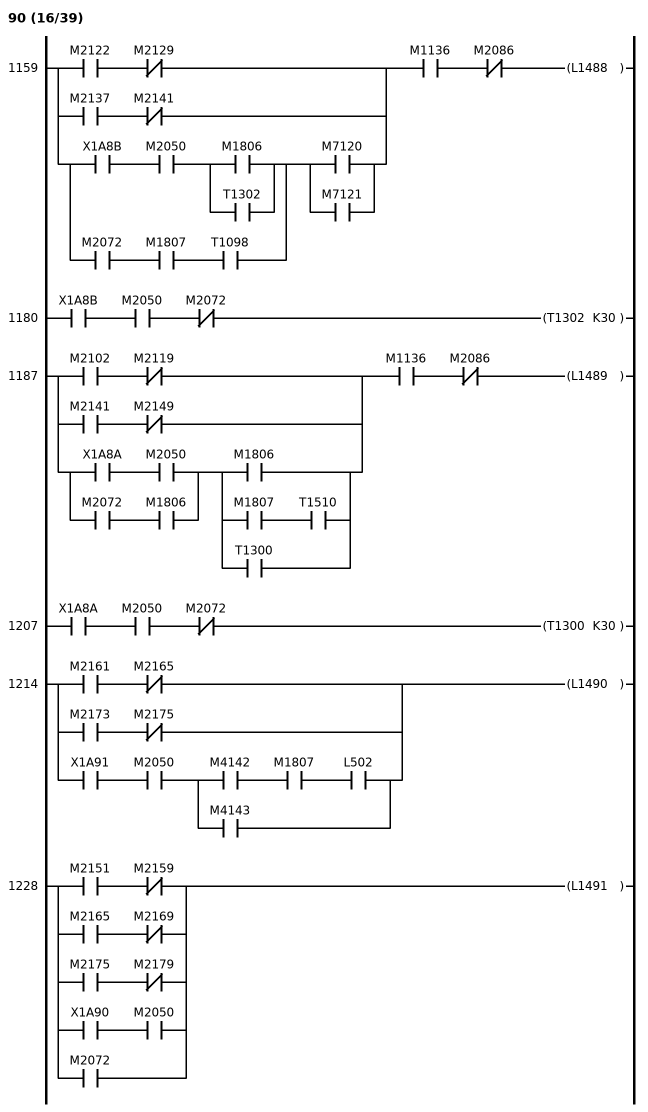
1159  LD      M2122
      ANI     M2129
      LD      M2137
      ANI     M2141
      ORB
      LD      X1A8B
      AND     M2050
      LD      M1806
      OR      T1302
      ANB
      LD      M2072
      AND     M1807
      AND     T1098
      ORB
      LD      M7120
      OR      M7121
      ANB
      ORB
      AND     M1136
      ANI     M2086
      OUT     L1488
1180  LD      X1A8B
      AND     M2050
      ANI     M2072
      OUT     T1302 K30
1187  LD      M2102
      ANI     M2119
      LD      M2141
      ANI     M2149
      ORB
      LD      X1A8A
      AND     M2050
      LD      M2072
      AND     M1806
      ORB
      LD      M1806
      LD      M1807
      AND     T1510
      ORB
      OR      T1300
      ANB
      ORB
      AND     M1136
      ANI     M2086
      OUT     L1489
1207  LD      X1A8A
      AND     M2050
      ANI     M2072
      OUT     T1300 K30
1214  LD      M2161
      ANI     M2165
      LD      M2173
      ANI     M2175
      ORB
      LD      X1A91
      AND     M2050
      LD      M4142
      AND     M1807
      AND     L502
      OR      M4143
      ANB
      ORB
      OUT     L1490
1228  LD      M2151
      ANI     M2159
      LD      M2165
      ANI     M2169
      ORB
      LD      M2175
      ANI     M2179
      ORB
      LD      X1A90
      AND     M2050
      ORB
      OR      M2072
      OUT     L1491
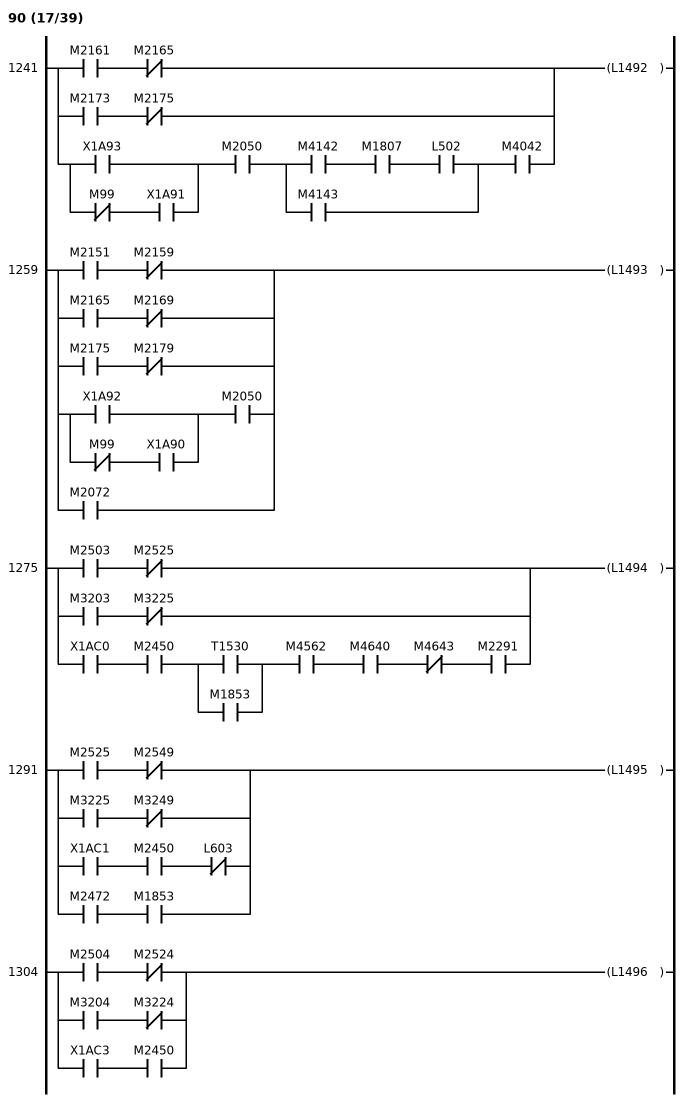
1241  LD      M2161
      ANI     M2165
      LD      M2173
      ANI     M2175
      ORB
      LD      X1A93
      LDI     M99
      AND     X1A91
      ORB
      AND     M2050
      LD      M4142
      AND     M1807
      AND     L502
      OR      M4143
      ANB
      AND     M4042
      ORB
      OUT     L1492
1259  LD      M2151
      ANI     M2159
      LD      M2165
      ANI     M2169
      ORB
      LD      M2175
      ANI     M2179
      ORB
      LD      X1A92
      LDI     M99
      AND     X1A90
      ORB
      AND     M2050
      ORB
      OR      M2072
      OUT     L1493
1275  LD      M2503
      ANI     M2525
      LD      M3203
      ANI     M3225
      ORB
      LD      X1AC0
      AND     M2450
      LD      T1530
      OR      M1853
      ANB
      AND     M4562
      AND     M4640
      ANI     M4643
      AND     M2291
      ORB
      OUT     L1494
1291  LD      M2525
      ANI     M2549
      LD      M3225
      ANI     M3249
      ORB
      LD      X1AC1
      AND     M2450
      ANI     L603
      ORB
      LD      M2472
      AND     M1853
      ORB
      OUT     L1495
1304  LD      M2504
      ANI     M2524
      LD      M3204
      ANI     M3224
      ORB
      LD      X1AC3
      AND     M2450
      ORB
      OUT     L1496
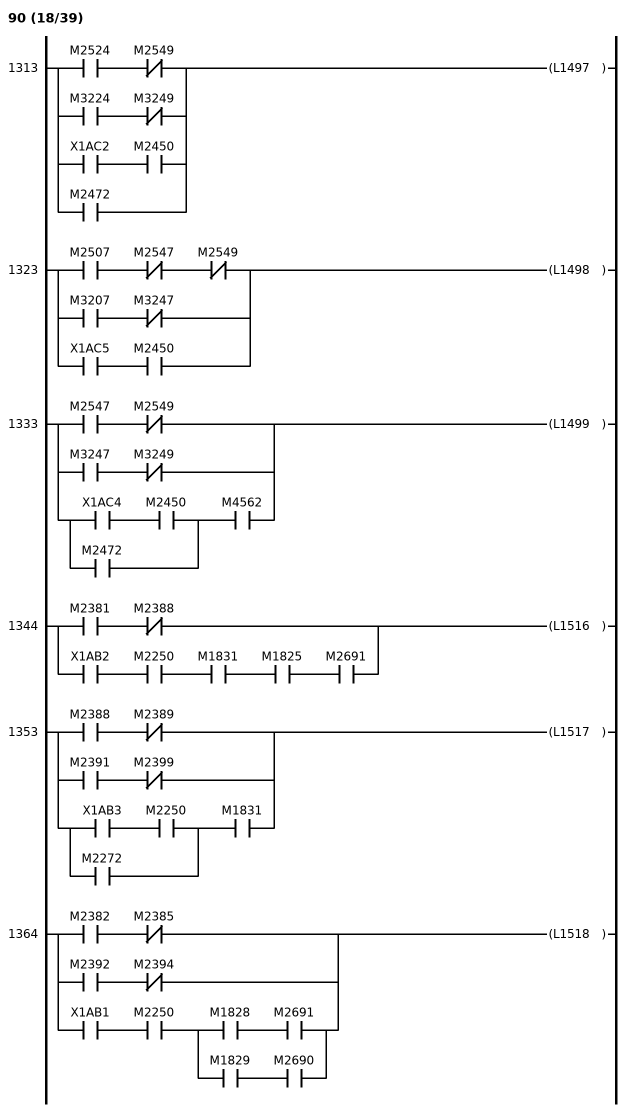
1313  LD      M2524
      ANI     M2549
      LD      M3224
      ANI     M3249
      ORB
      LD      X1AC2
      AND     M2450
      ORB
      OR      M2472
      OUT     L1497
1323  LD      M2507
      ANI     M2547
      ANI     M2549
      LD      M3207
      ANI     M3247
      ORB
      LD      X1AC5
      AND     M2450
      ORB
      OUT     L1498
1333  LD      M2547
      ANI     M2549
      LD      M3247
      ANI     M3249
      ORB
      LD      X1AC4
      AND     M2450
      OR      M2472
      AND     M4562
      ORB
      OUT     L1499
1344  LD      M2381
      ANI     M2388
      LD      X1AB2
      AND     M2250
      AND     M1831
      AND     M1825
      AND     M2691
      ORB
      OUT     L1516
1353  LD      M2388
      ANI     M2389
      LD      M2391
      ANI     M2399
      ORB
      LD      X1AB3
      AND     M2250
      OR      M2272
      AND     M1831
      ORB
      OUT     L1517
1364  LD      M2382
      ANI     M2385
      LD      M2392
      ANI     M2394
      ORB
      LD      X1AB1
      AND     M2250
      LD      M1828
      AND     M2691
      LD      M1829
      AND     M2690
      ORB
      ANB
      ORB
      OUT     L1518
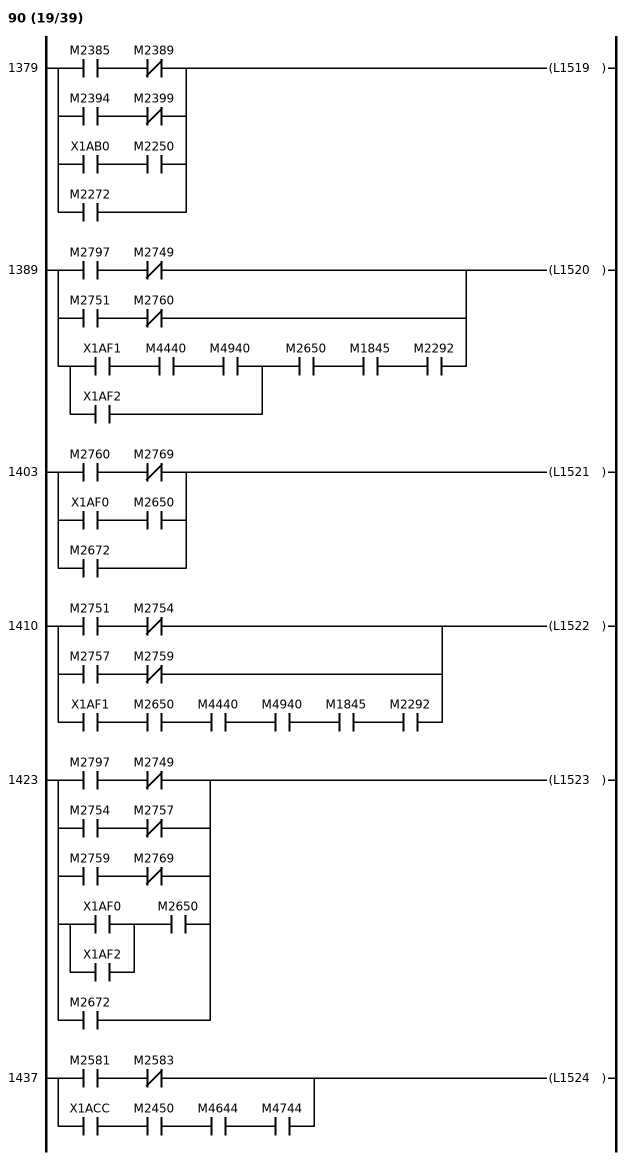
1379  LD      M2385
      ANI     M2389
      LD      M2394
      ANI     M2399
      ORB
      LD      X1AB0
      AND     M2250
      ORB
      OR      M2272
      OUT     L1519
1389  LD      M2797
      ANI     M2749
      LD      M2751
      ANI     M2760
      ORB
      LD      X1AF1
      AND     M4440
      AND     M4940
      OR      X1AF2
      AND     M2650
      AND     M1845
      AND     M2292
      ORB
      OUT     L1520
1403  LD      M2760
      ANI     M2769
      LD      X1AF0
      AND     M2650
      ORB
      OR      M2672
      OUT     L1521
1410  LD      M2751
      ANI     M2754
      LD      M2757
      ANI     M2759
      ORB
      LD      X1AF1
      AND     M2650
      AND     M4440
      AND     M4940
      AND     M1845
      AND     M2292
      ORB
      OUT     L1522
1423  LD      M2797
      ANI     M2749
      LD      M2754
      ANI     M2757
      ORB
      LD      M2759
      ANI     M2769
      ORB
      LD      X1AF0
      OR      X1AF2
      AND     M2650
      ORB
      OR      M2672
      OUT     L1523
1437  LD      M2581
      ANI     M2583
      LD      X1ACC
      AND     M2450
      AND     M4644
      AND     M4744
      ORB
      OUT     L1524
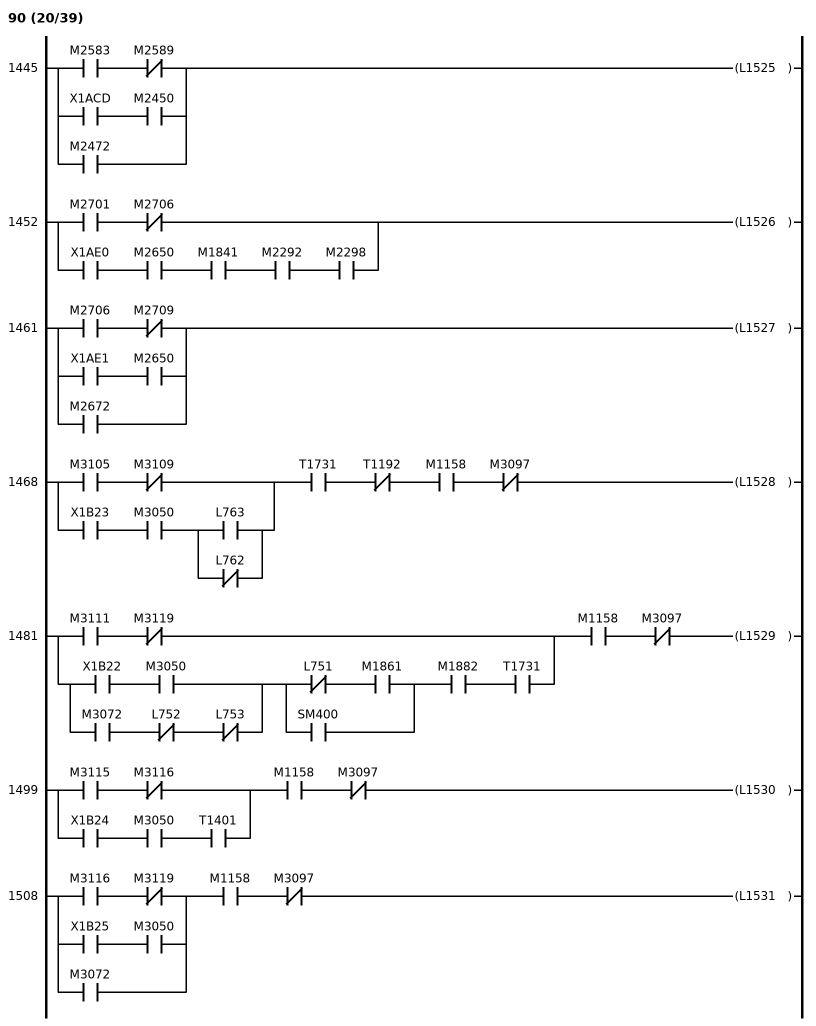
1445  LD      M2583
      ANI     M2589
      LD      X1ACD
      AND     M2450
      ORB
      OR      M2472
      OUT     L1525
1452  LD      M2701
      ANI     M2706
      LD      X1AE0
      AND     M2650
      AND     M1841
      AND     M2292
      AND     M2298
      ORB
      OUT     L1526
1461  LD      M2706
      ANI     M2709
      LD      X1AE1
      AND     M2650
      ORB
      OR      M2672
      OUT     L1527
1468  LD      M3105
      ANI     M3109
      LD      X1B23
      AND     M3050
      LD      L763
      ORI     L762
      ANB
      ORB
      AND     T1731
      ANI     T1192
      AND     M1158
      ANI     M3097
      OUT     L1528
1481  LD      M3111
      ANI     M3119
      LD      X1B22
      AND     M3050
      LD      M3072
      ANI     L752
      ANI     L753
      ORB
      LDI     L751
      AND     M1861
      OR      SM400
      ANB
      AND     M1882
      AND     T1731
      ORB
      AND     M1158
      ANI     M3097
      OUT     L1529
1499  LD      M3115
      ANI     M3116
      LD      X1B24
      AND     M3050
      AND     T1401
      ORB
      AND     M1158
      ANI     M3097
      OUT     L1530
1508  LD      M3116
      ANI     M3119
      LD      X1B25
      AND     M3050
      ORB
      OR      M3072
      AND     M1158
      ANI     M3097
      OUT     L1531
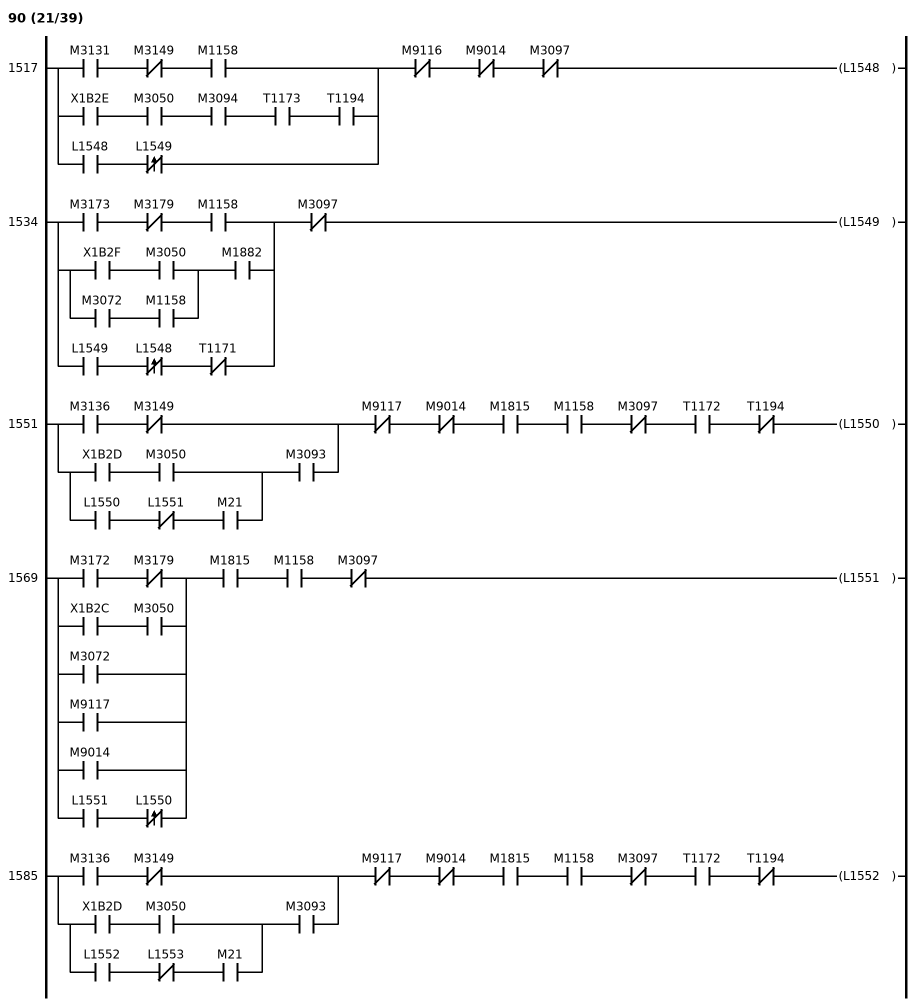
1517  LD      M3131
      ANI     M3149
      AND     M1158
      LD      X1B2E
      AND     M3050
      AND     M3094
      AND     T1173
      AND     T1194
      ORB
      LD      L1548
      ANDPI   L1549
      ORB
      ANI     M9116
      ANI     M9014
      ANI     M3097
      OUT     L1548
1534  LD      M3173
      ANI     M3179
      AND     M1158
      LD      X1B2F
      AND     M3050
      LD      M3072
      AND     M1158
      ORB
      AND     M1882
      ORB
      LD      L1549
      ANDPI   L1548
      ANI     T1171
      ORB
      ANI     M3097
      OUT     L1549
1551  LD      M3136
      ANI     M3149
      LD      X1B2D
      AND     M3050
      LD      L1550
      ANI     L1551
      AND     M21
      ORB
      AND     M3093
      ORB
      ANI     M9117
      ANI     M9014
      AND     M1815
      AND     M1158
      ANI     M3097
      AND     T1172
      ANI     T1194
      OUT     L1550
1569  LD      M3172
      ANI     M3179
      LD      X1B2C
      AND     M3050
      ORB
      OR      M3072
      OR      M9117
      OR      M9014
      LD      L1551
      ANDPI   L1550
      ORB
      AND     M1815
      AND     M1158
      ANI     M3097
      OUT     L1551
1585  LD      M3136
      ANI     M3149
      LD      X1B2D
      AND     M3050
      LD      L1552
      ANI     L1553
      AND     M21
      ORB
      AND     M3093
      ORB
      ANI     M9117
      ANI     M9014
      AND     M1815
      AND     M1158
      ANI     M3097
      AND     T1172
      ANI     T1194
      OUT     L1552
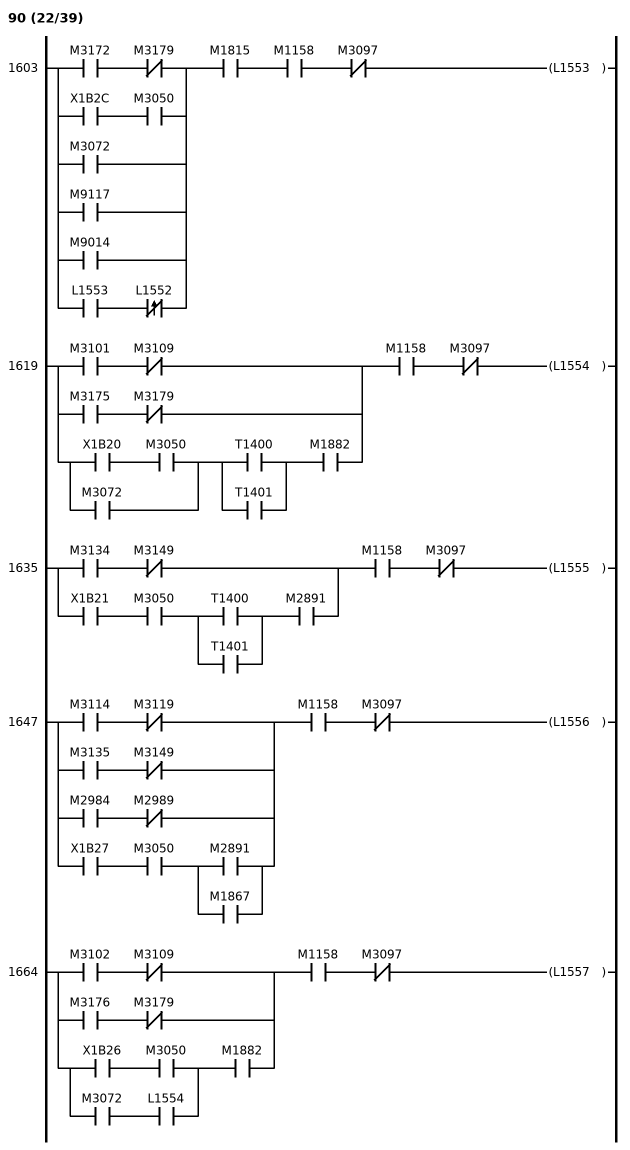
1603  LD      M3172
      ANI     M3179
      LD      X1B2C
      AND     M3050
      ORB
      OR      M3072
      OR      M9117
      OR      M9014
      LD      L1553
      ANDPI   L1552
      ORB
      AND     M1815
      AND     M1158
      ANI     M3097
      OUT     L1553
1619  LD      M3101
      ANI     M3109
      LD      M3175
      ANI     M3179
      ORB
      LD      X1B20
      AND     M3050
      OR      M3072
      LD      T1400
      OR      T1401
      ANB
      AND     M1882
      ORB
      AND     M1158
      ANI     M3097
      OUT     L1554
1635  LD      M3134
      ANI     M3149
      LD      X1B21
      AND     M3050
      LD      T1400
      OR      T1401
      ANB
      AND     M2891
      ORB
      AND     M1158
      ANI     M3097
      OUT     L1555
1647  LD      M3114
      ANI     M3119
      LD      M3135
      ANI     M3149
      ORB
      LD      M2984
      ANI     M2989
      ORB
      LD      X1B27
      AND     M3050
      LD      M2891
      OR      M1867
      ANB
      ORB
      AND     M1158
      ANI     M3097
      OUT     L1556
1664  LD      M3102
      ANI     M3109
      LD      M3176
      ANI     M3179
      ORB
      LD      X1B26
      AND     M3050
      LD      M3072
      AND     L1554
      ORB
      AND     M1882
      ORB
      AND     M1158
      ANI     M3097
      OUT     L1557
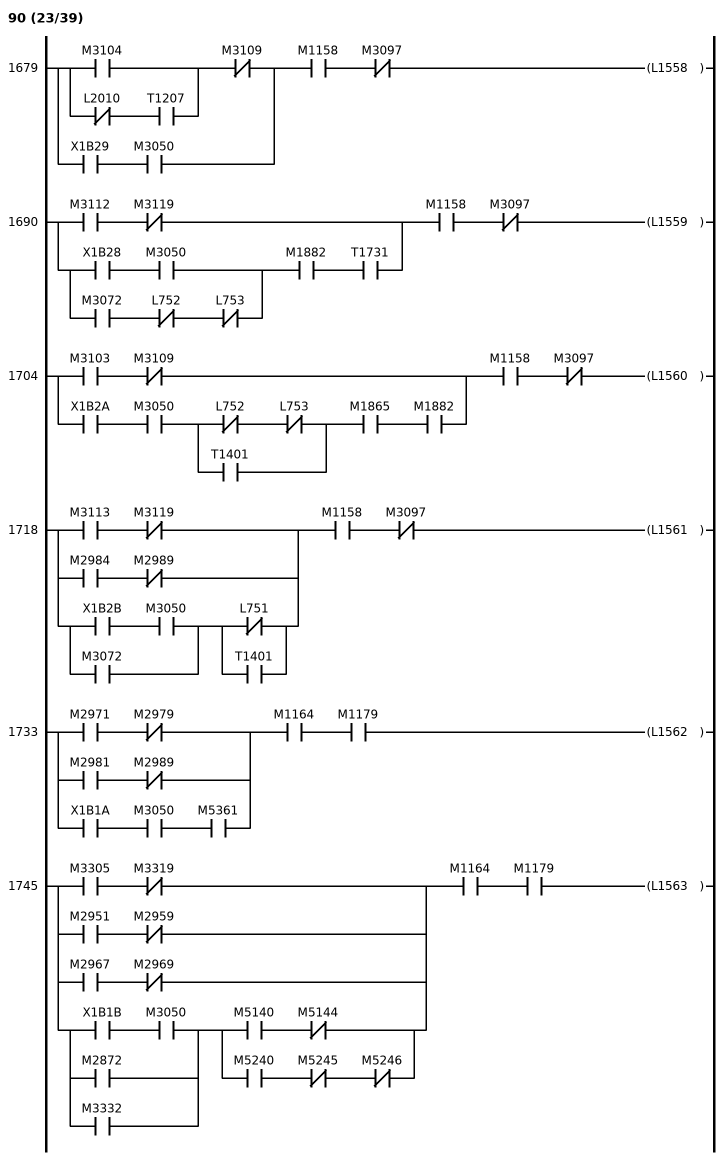
1679  LD      M3104
      LDI     L2010
      AND     T1207
      ORB
      ANI     M3109
      LD      X1B29
      AND     M3050
      ORB
      AND     M1158
      ANI     M3097
      OUT     L1558
1690  LD      M3112
      ANI     M3119
      LD      X1B28
      AND     M3050
      LD      M3072
      ANI     L752
      ANI     L753
      ORB
      AND     M1882
      AND     T1731
      ORB
      AND     M1158
      ANI     M3097
      OUT     L1559
1704  LD      M3103
      ANI     M3109
      LD      X1B2A
      AND     M3050
      LDI     L752
      ANI     L753
      OR      T1401
      ANB
      AND     M1865
      AND     M1882
      ORB
      AND     M1158
      ANI     M3097
      OUT     L1560
1718  LD      M3113
      ANI     M3119
      LD      M2984
      ANI     M2989
      ORB
      LD      X1B2B
      AND     M3050
      OR      M3072
      LDI     L751
      OR      T1401
      ANB
      ORB
      AND     M1158
      ANI     M3097
      OUT     L1561
1733  LD      M2971
      ANI     M2979
      LD      M2981
      ANI     M2989
      ORB
      LD      X1B1A
      AND     M3050
      AND     M5361
      ORB
      AND     M1164
      AND     M1179
      OUT     L1562
1745  LD      M3305
      ANI     M3319
      LD      M2951
      ANI     M2959
      ORB
      LD      M2967
      ANI     M2969
      ORB
      LD      X1B1B
      AND     M3050
      OR      M2872
      OR      M3332
      LD      M5140
      ANI     M5144
      LD      M5240
      ANI     M5245
      ANI     M5246
      ORB
      ANB
      ORB
      AND     M1164
      AND     M1179
      OUT     L1563
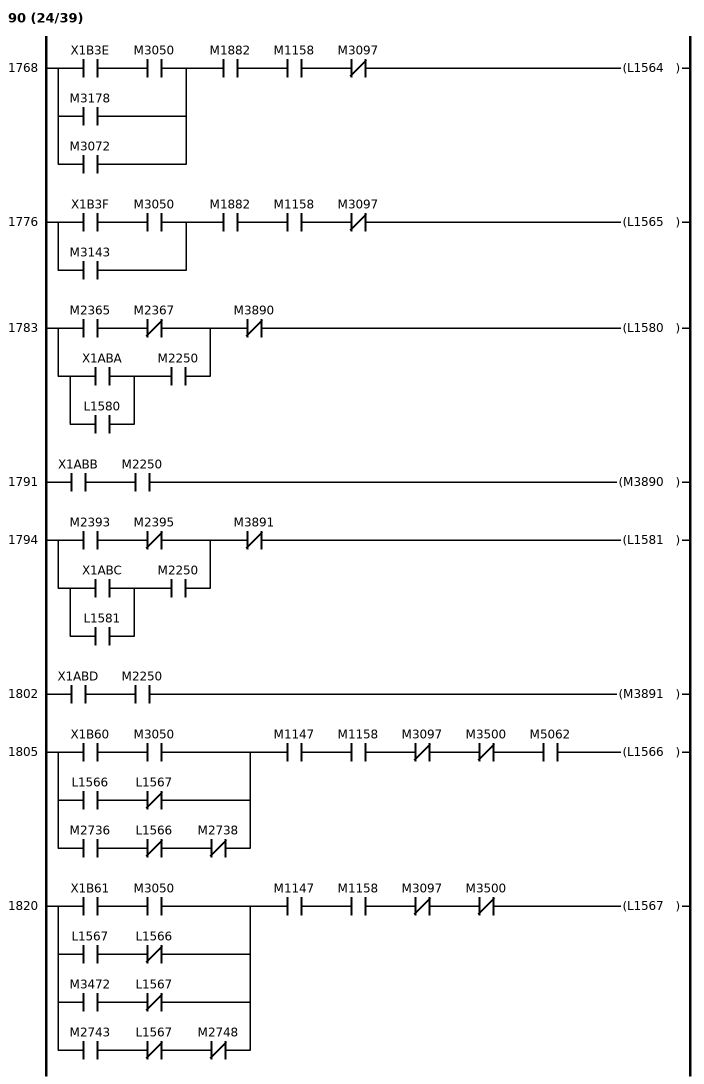
1768  LD      X1B3E
      AND     M3050
      OR      M3178
      OR      M3072
      AND     M1882
      AND     M1158
      ANI     M3097
      OUT     L1564
1776  LD      X1B3F
      AND     M3050
      OR      M3143
      AND     M1882
      AND     M1158
      ANI     M3097
      OUT     L1565
1783  LD      M2365
      ANI     M2367
      LD      X1ABA
      OR      L1580
      AND     M2250
      ORB
      ANI     M3890
      OUT     L1580
1791  LD      X1ABB
      AND     M2250
      OUT     M3890
1794  LD      M2393
      ANI     M2395
      LD      X1ABC
      OR      L1581
      AND     M2250
      ORB
      ANI     M3891
      OUT     L1581
1802  LD      X1ABD
      AND     M2250
      OUT     M3891
1805  LD      X1B60
      AND     M3050
      LD      L1566
      ANI     L1567
      ORB
      LD      M2736
      ANI     L1566
      ANI     M2738
      ORB
      AND     M1147
      AND     M1158
      ANI     M3097
      ANI     M3500
      AND     M5062
      OUT     L1566
1820  LD      X1B61
      AND     M3050
      LD      L1567
      ANI     L1566
      ORB
      LD      M3472
      ANI     L1567
      ORB
      LD      M2743
      ANI     L1567
      ANI     M2748
      ORB
      AND     M1147
      AND     M1158
      ANI     M3097
      ANI     M3500
      OUT     L1567
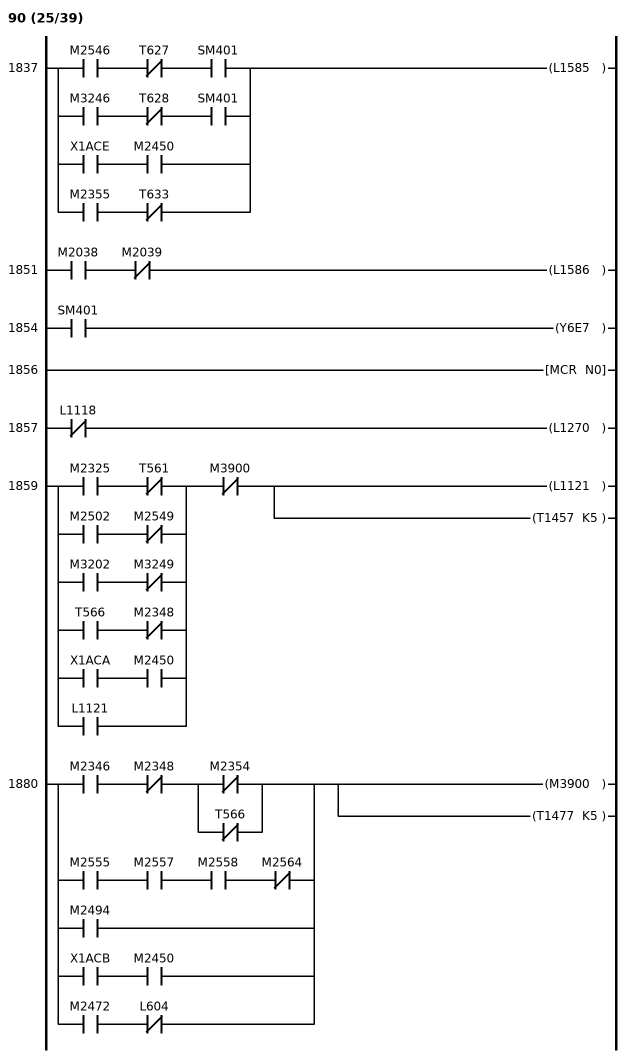
1837  LD      M2546
      ANI     T627
      AND     SM401
      LD      M3246
      ANI     T628
      AND     SM401
      ORB
      LD      X1ACE
      AND     M2450
      ORB
      LD      M2355
      ANI     T633
      ORB
      OUT     L1585
1851  LD      M2038
      ANI     M2039
      OUT     L1586
1854  LD      SM401
      OUT     Y6E7
1856  MCR     N0
1857  LDI     L1118
      OUT     L1270
1859  LD      M2325
      ANI     T561
      LD      M2502
      ANI     M2549
      ORB
      LD      M3202
      ANI     M3249
      ORB
      LD      T566
      ANI     M2348
      ORB
      LD      X1ACA
      AND     M2450
      ORB
      OR      L1121
      ANI     M3900
      OUT     L1121
      OUT     T1457 K5
1880  LD      M2346
      ANI     M2348
      LDI     M2354
      ORI     T566
      ANB
      LD      M2555
      AND     M2557
      AND     M2558
      ANI     M2564
      ORB
      OR      M2494
      LD      X1ACB
      AND     M2450
      ORB
      LD      M2472
      ANI     L604
      ORB
      OUT     M3900
      OUT     T1477 K5
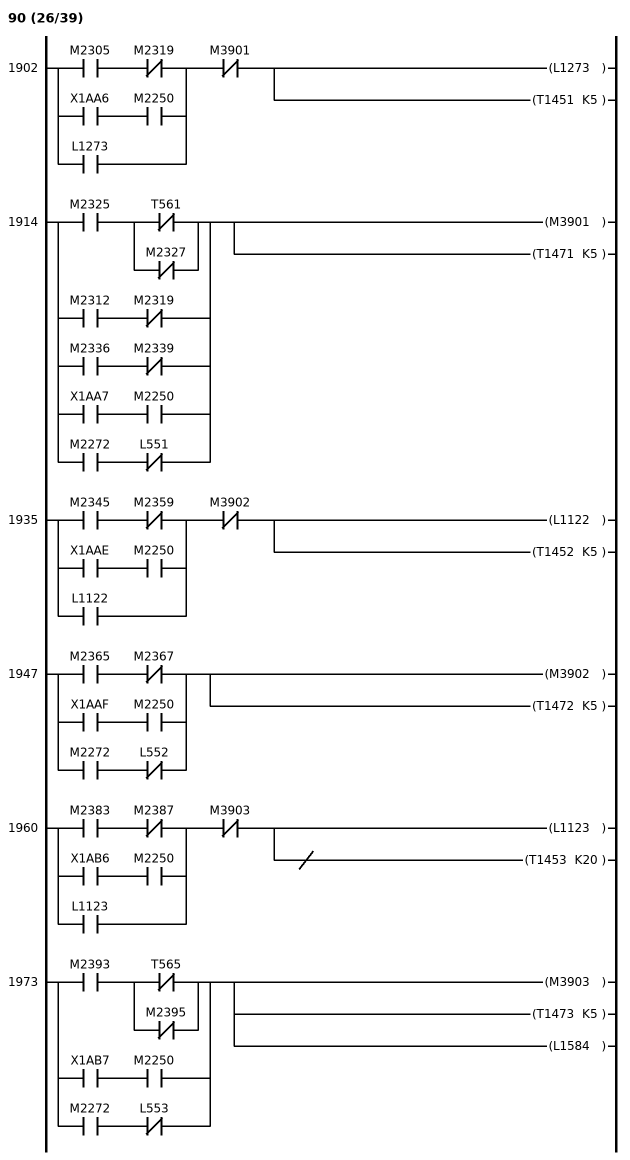
1902  LD      M2305
      ANI     M2319
      LD      X1AA6
      AND     M2250
      ORB
      OR      L1273
      ANI     M3901
      OUT     L1273
      OUT     T1451 K5
1914  LD      M2325
      LDI     T561
      ORI     M2327
      ANB
      LD      M2312
      ANI     M2319
      ORB
      LD      M2336
      ANI     M2339
      ORB
      LD      X1AA7
      AND     M2250
      ORB
      LD      M2272
      ANI     L551
      ORB
      OUT     M3901
      OUT     T1471 K5
1935  LD      M2345
      ANI     M2359
      LD      X1AAE
      AND     M2250
      ORB
      OR      L1122
      ANI     M3902
      OUT     L1122
      OUT     T1452 K5
1947  LD      M2365
      ANI     M2367
      LD      X1AAF
      AND     M2250
      ORB
      LD      M2272
      ANI     L552
      ORB
      OUT     M3902
      OUT     T1472 K5
1960  LD      M2383
      ANI     M2387
      LD      X1AB6
      AND     M2250
      ORB
      OR      L1123
      ANI     M3903
      OUT     L1123
      INV
      OUT     T1453 K20
1973  LD      M2393
      LDI     T565
      ORI     M2395
      ANB
      LD      X1AB7
      AND     M2250
      ORB
      LD      M2272
      ANI     L553
      ORB
      OUT     M3903
      OUT     T1473 K5
      OUT     L1584
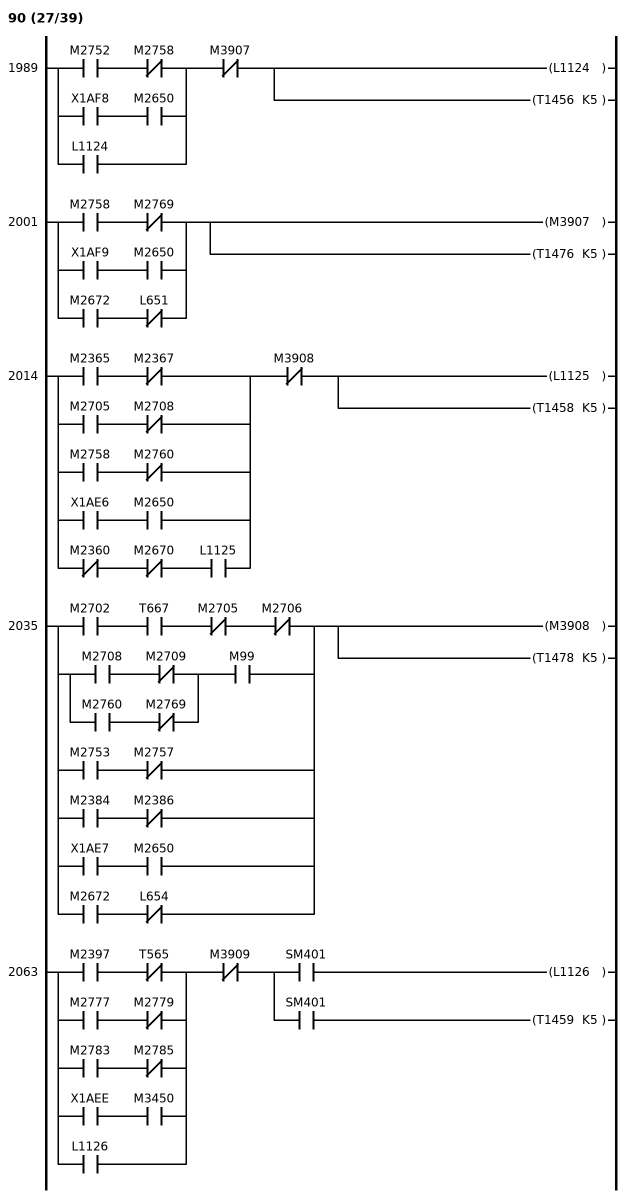
1989  LD      M2752
      ANI     M2758
      LD      X1AF8
      AND     M2650
      ORB
      OR      L1124
      ANI     M3907
      OUT     L1124
      OUT     T1456 K5
2001  LD      M2758
      ANI     M2769
      LD      X1AF9
      AND     M2650
      ORB
      LD      M2672
      ANI     L651
      ORB
      OUT     M3907
      OUT     T1476 K5
2014  LD      M2365
      ANI     M2367
      LD      M2705
      ANI     M2708
      ORB
      LD      M2758
      ANI     M2760
      ORB
      LD      X1AE6
      AND     M2650
      ORB
      LDI     M2360
      ANI     M2670
      AND     L1125
      ORB
      ANI     M3908
      OUT     L1125
      OUT     T1458 K5
2035  LD      M2702
      AND     T667
      ANI     M2705
      ANI     M2706
      LD      M2708
      ANI     M2709
      LD      M2760
      ANI     M2769
      ORB
      AND     M99
      ORB
      LD      M2753
      ANI     M2757
      ORB
      LD      M2384
      ANI     M2386
      ORB
      LD      X1AE7
      AND     M2650
      ORB
      LD      M2672
      ANI     L654
      ORB
      OUT     M3908
      OUT     T1478 K5
2063  LD      M2397
      ANI     T565
      LD      M2777
      ANI     M2779
      ORB
      LD      M2783
      ANI     M2785
      ORB
      LD      X1AEE
      AND     M3450
      ORB
      OR      L1126
      ANI     M3909
      MPS
      AND     SM401
      OUT     L1126
      MPP
      AND     SM401
      OUT     T1459 K5
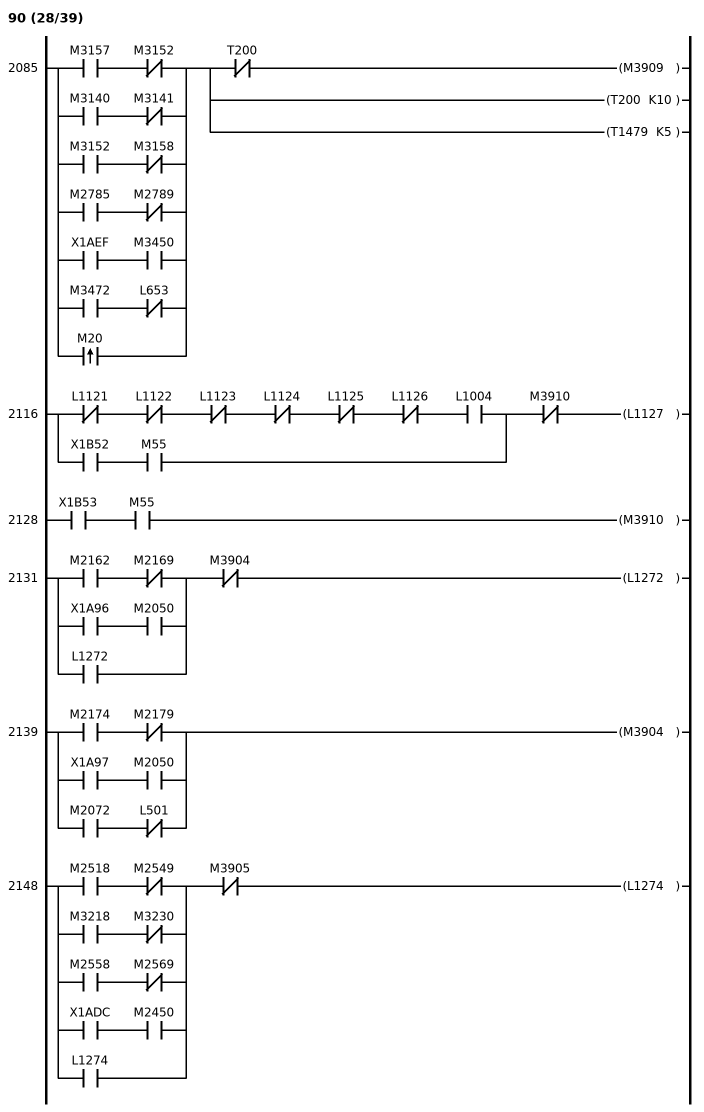
2085  LD      M3157
      ANI     M3152
      LD      M3140
      ANI     M3141
      ORB
      LD      M3152
      ANI     M3158
      ORB
      LD      M2785
      ANI     M2789
      ORB
      LD      X1AEF
      AND     M3450
      ORB
      LD      M3472
      ANI     L653
      ORB
      ORP     M20
      MPS
      ANI     T200
      OUT     M3909
      MPP
      OUT     T200 K10
      OUT     T1479 K5
2116  LDI     L1121
      ANI     L1122
      ANI     L1123
      ANI     L1124
      ANI     L1125
      ANI     L1126
      AND     L1004
      LD      X1B52
      AND     M55
      ORB
      ANI     M3910
      OUT     L1127
2128  LD      X1B53
      AND     M55
      OUT     M3910
2131  LD      M2162
      ANI     M2169
      LD      X1A96
      AND     M2050
      ORB
      OR      L1272
      ANI     M3904
      OUT     L1272
2139  LD      M2174
      ANI     M2179
      LD      X1A97
      AND     M2050
      ORB
      LD      M2072
      ANI     L501
      ORB
      OUT     M3904
2148  LD      M2518
      ANI     M2549
      LD      M3218
      ANI     M3230
      ORB
      LD      M2558
      ANI     M2569
      ORB
      LD      X1ADC
      AND     M2450
      ORB
      OR      L1274
      ANI     M3905
      OUT     L1274
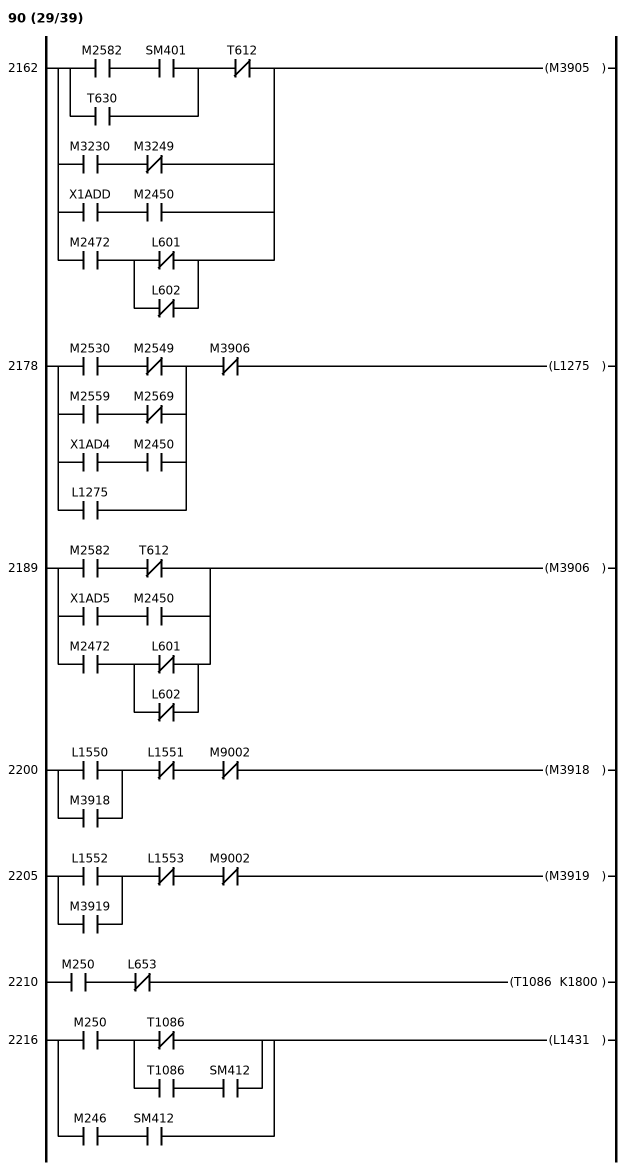
2162  LD      M2582
      AND     SM401
      OR      T630
      ANI     T612
      LD      M3230
      ANI     M3249
      ORB
      LD      X1ADD
      AND     M2450
      ORB
      LD      M2472
      LDI     L601
      ORI     L602
      ANB
      ORB
      OUT     M3905
2178  LD      M2530
      ANI     M2549
      LD      M2559
      ANI     M2569
      ORB
      LD      X1AD4
      AND     M2450
      ORB
      OR      L1275
      ANI     M3906
      OUT     L1275
2189  LD      M2582
      ANI     T612
      LD      X1AD5
      AND     M2450
      ORB
      LD      M2472
      LDI     L601
      ORI     L602
      ANB
      ORB
      OUT     M3906
2200  LD      L1550
      OR      M3918
      ANI     L1551
      ANI     M9002
      OUT     M3918
2205  LD      L1552
      OR      M3919
      ANI     L1553
      ANI     M9002
      OUT     M3919
2210  LD      M250
      ANI     L653
      OUT     T1086 K1800
2216  LD      M250
      LDI     T1086
      LD      T1086
      AND     SM412
      ORB
      ANB
      LD      M246
      AND     SM412
      ORB
      OUT     L1431
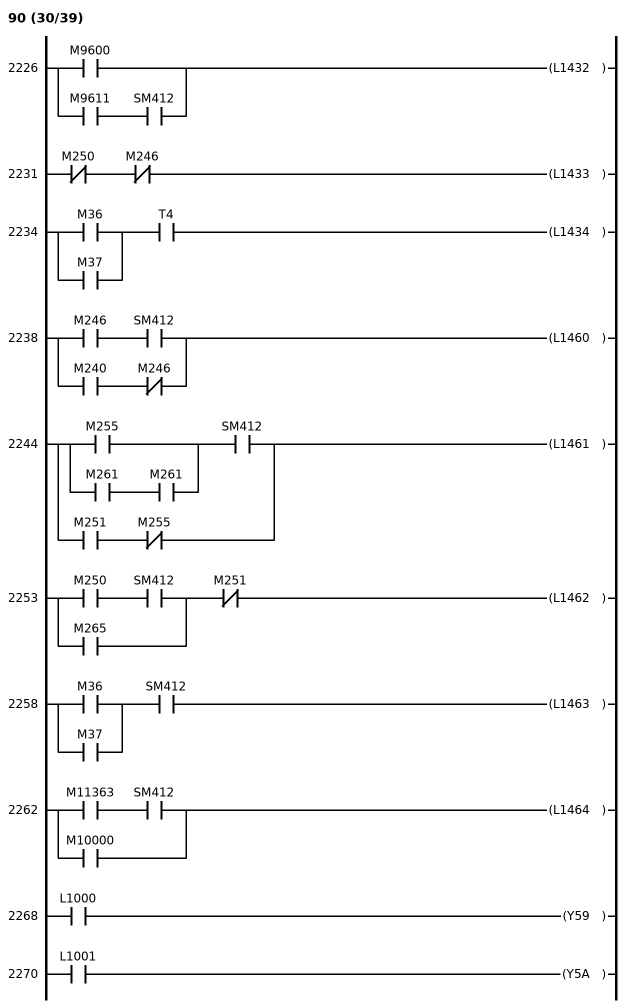
2226  LD      M9600
      LD      M9611
      AND     SM412
      ORB
      OUT     L1432
2231  LDI     M250
      ANI     M246
      OUT     L1433
2234  LD      M36
      OR      M37
      AND     T4
      OUT     L1434
2238  LD      M246
      AND     SM412
      LD      M240
      ANI     M246
      ORB
      OUT     L1460
2244  LD      M255
      LD      M261
      AND     M261
      ORB
      AND     SM412
      LD      M251
      ANI     M255
      ORB
      OUT     L1461
2253  LD      M250
      AND     SM412
      OR      M265
      ANI     M251
      OUT     L1462
2258  LD      M36
      OR      M37
      AND     SM412
      OUT     L1463
2262  LD      M11363
      AND     SM412
      OR      M10000
      OUT     L1464
; 
2268  LD      L1000
      OUT     Y59
2270  LD      L1001
      OUT     Y5A
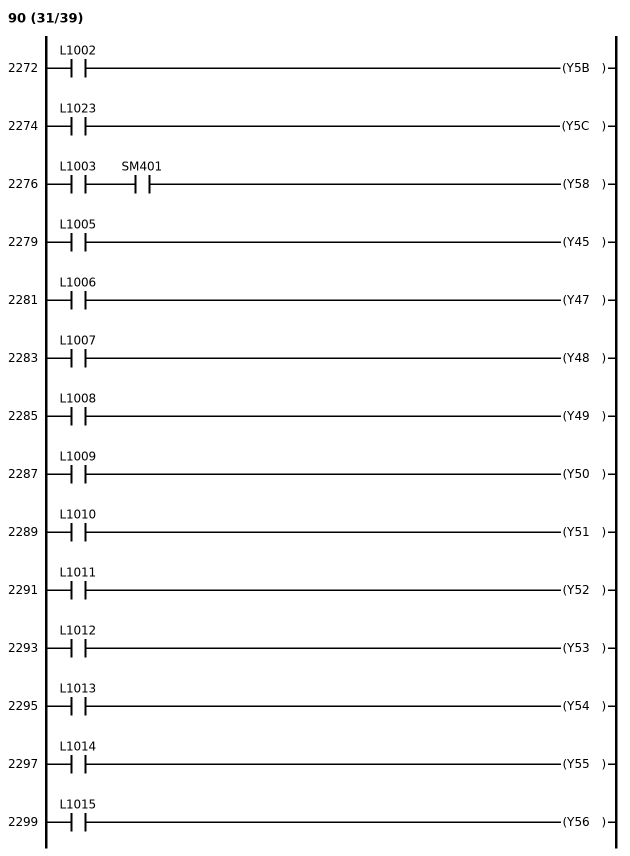
2272  LD      L1002
      OUT     Y5B
2274  LD      L1023
      OUT     Y5C
2276  LD      L1003
      AND     SM401
      OUT     Y58
2279  LD      L1005
      OUT     Y45
2281  LD      L1006
      OUT     Y47
2283  LD      L1007
      OUT     Y48
2285  LD      L1008
      OUT     Y49
2287  LD      L1009
      OUT     Y50
2289  LD      L1010
      OUT     Y51
2291  LD      L1011
      OUT     Y52
2293  LD      L1012
      OUT     Y53
2295  LD      L1013
      OUT     Y54
2297  LD      L1014
      OUT     Y55
2299  LD      L1015
      OUT     Y56
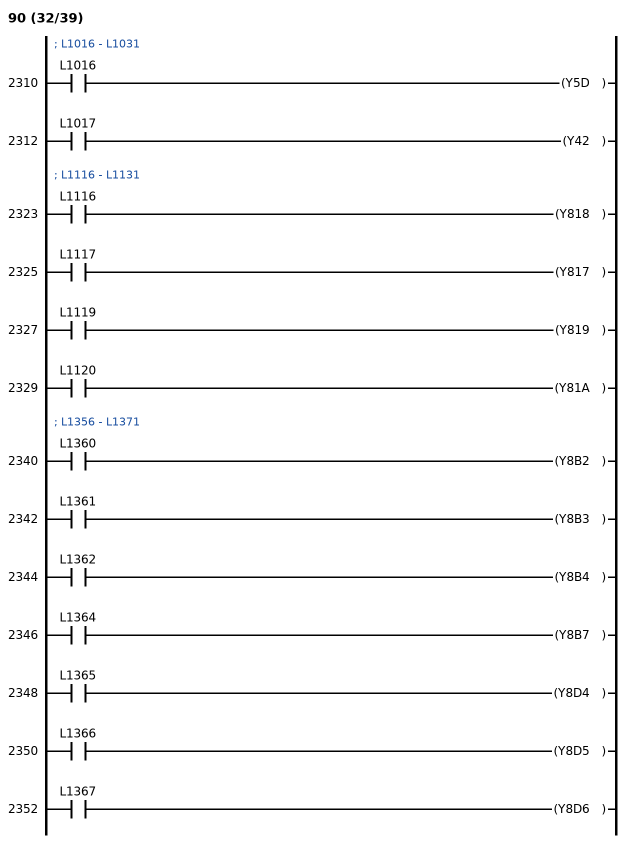
; L1016 - L1031
2310  LD      L1016
      OUT     Y5D
2312  LD      L1017
      OUT     Y42
; L1116 - L1131
2323  LD      L1116
      OUT     Y818
2325  LD      L1117
      OUT     Y817
2327  LD      L1119
      OUT     Y819
2329  LD      L1120
      OUT     Y81A
; L1356 - L1371
2340  LD      L1360
      OUT     Y8B2
2342  LD      L1361
      OUT     Y8B3
2344  LD      L1362
      OUT     Y8B4
2346  LD      L1364
      OUT     Y8B7
2348  LD      L1365
      OUT     Y8D4
2350  LD      L1366
      OUT     Y8D5
2352  LD      L1367
      OUT     Y8D6
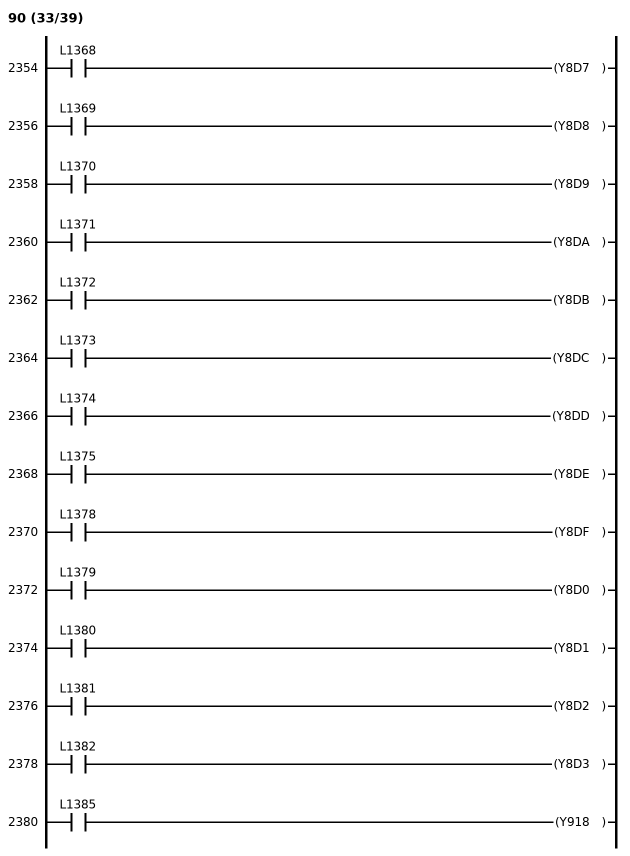
2354  LD      L1368
      OUT     Y8D7
2356  LD      L1369
      OUT     Y8D8
2358  LD      L1370
      OUT     Y8D9
2360  LD      L1371
      OUT     Y8DA
2362  LD      L1372
      OUT     Y8DB
2364  LD      L1373
      OUT     Y8DC
2366  LD      L1374
      OUT     Y8DD
2368  LD      L1375
      OUT     Y8DE
2370  LD      L1378
      OUT     Y8DF
2372  LD      L1379
      OUT     Y8D0
2374  LD      L1380
      OUT     Y8D1
2376  LD      L1381
      OUT     Y8D2
2378  LD      L1382
      OUT     Y8D3
2380  LD      L1385
      OUT     Y918
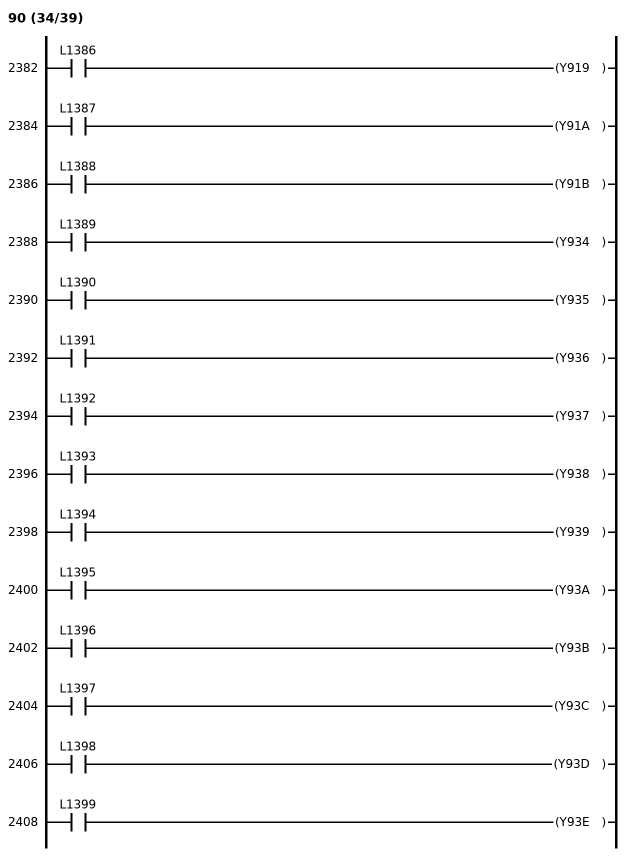
2382  LD      L1386
      OUT     Y919
2384  LD      L1387
      OUT     Y91A
2386  LD      L1388
      OUT     Y91B
2388  LD      L1389
      OUT     Y934
2390  LD      L1390
      OUT     Y935
2392  LD      L1391
      OUT     Y936
2394  LD      L1392
      OUT     Y937
2396  LD      L1393
      OUT     Y938
2398  LD      L1394
      OUT     Y939
2400  LD      L1395
      OUT     Y93A
2402  LD      L1396
      OUT     Y93B
2404  LD      L1397
      OUT     Y93C
2406  LD      L1398
      OUT     Y93D
2408  LD      L1399
      OUT     Y93E
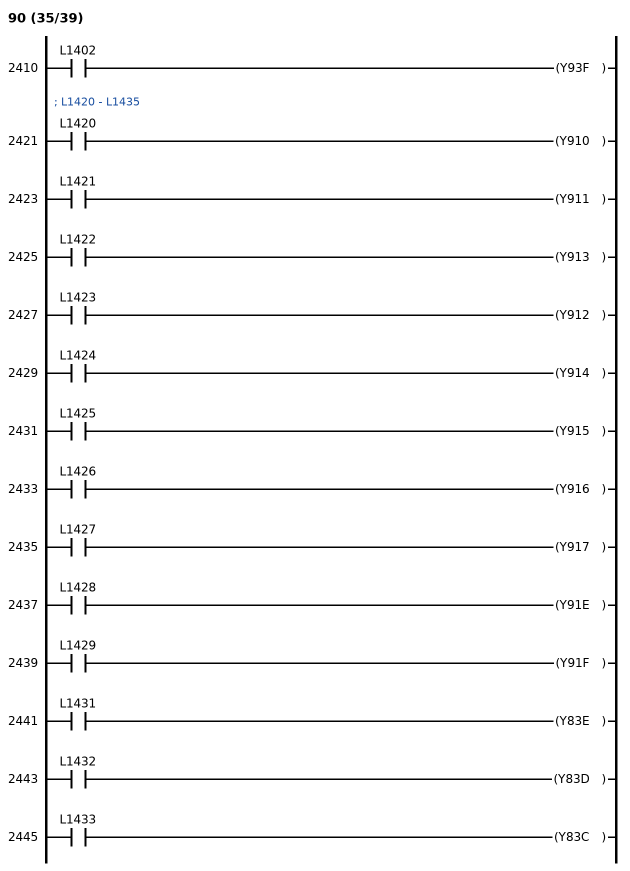
2410  LD      L1402
      OUT     Y93F
; L1420 - L1435
2421  LD      L1420
      OUT     Y910
2423  LD      L1421
      OUT     Y911
2425  LD      L1422
      OUT     Y913
2427  LD      L1423
      OUT     Y912
2429  LD      L1424
      OUT     Y914
2431  LD      L1425
      OUT     Y915
2433  LD      L1426
      OUT     Y916
2435  LD      L1427
      OUT     Y917
2437  LD      L1428
      OUT     Y91E
2439  LD      L1429
      OUT     Y91F
2441  LD      L1431
      OUT     Y83E
2443  LD      L1432
      OUT     Y83D
2445  LD      L1433
      OUT     Y83C
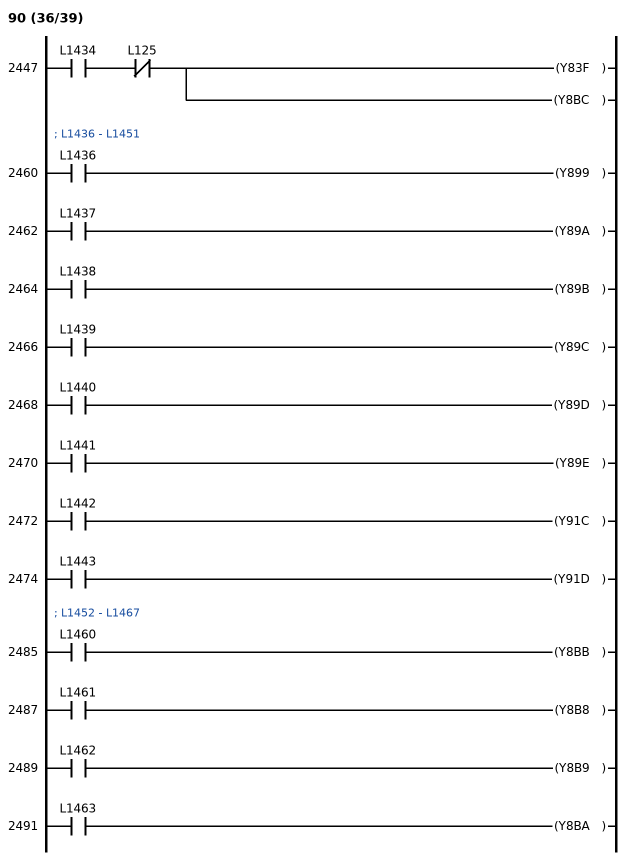
2447  LD      L1434
      ANI     L125
      OUT     Y83F
      OUT     Y8BC
; L1436 - L1451
2460  LD      L1436
      OUT     Y899
2462  LD      L1437
      OUT     Y89A
2464  LD      L1438
      OUT     Y89B
2466  LD      L1439
      OUT     Y89C
2468  LD      L1440
      OUT     Y89D
2470  LD      L1441
      OUT     Y89E
2472  LD      L1442
      OUT     Y91C
2474  LD      L1443
      OUT     Y91D
; L1452 - L1467
2485  LD      L1460
      OUT     Y8BB
2487  LD      L1461
      OUT     Y8B8
2489  LD      L1462
      OUT     Y8B9
2491  LD      L1463
      OUT     Y8BA
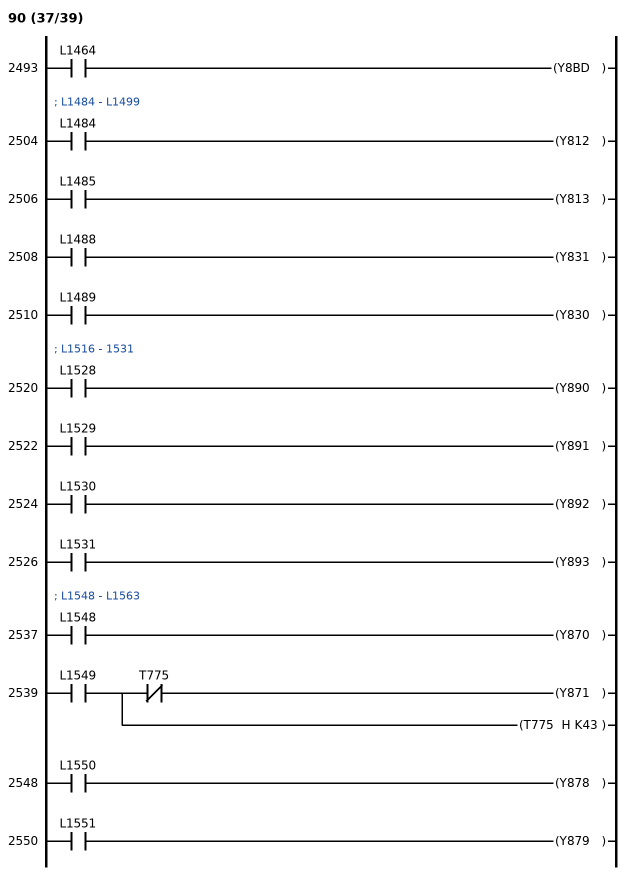
2493  LD      L1464
      OUT     Y8BD
; L1484 - L1499
2504  LD      L1484
      OUT     Y812
2506  LD      L1485
      OUT     Y813
2508  LD      L1488
      OUT     Y831
2510  LD      L1489
      OUT     Y830
; L1516 - 1531
2520  LD      L1528
      OUT     Y890
2522  LD      L1529
      OUT     Y891
2524  LD      L1530
      OUT     Y892
2526  LD      L1531
      OUT     Y893
; L1548 - L1563
2537  LD      L1548
      OUT     Y870
2539  LD      L1549
      MPS
      ANI     T775
      OUT     Y871
      MPP
      OUTH    T775 K43
2548  LD      L1550
      OUT     Y878
2550  LD      L1551
      OUT     Y879
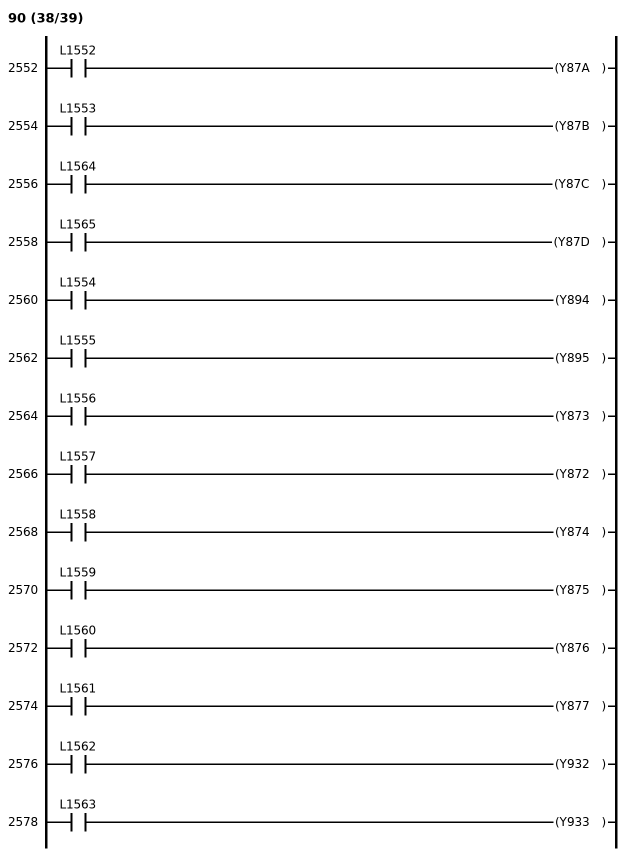
2552  LD      L1552
      OUT     Y87A
2554  LD      L1553
      OUT     Y87B
2556  LD      L1564
      OUT     Y87C
2558  LD      L1565
      OUT     Y87D
2560  LD      L1554
      OUT     Y894
2562  LD      L1555
      OUT     Y895
2564  LD      L1556
      OUT     Y873
2566  LD      L1557
      OUT     Y872
2568  LD      L1558
      OUT     Y874
2570  LD      L1559
      OUT     Y875
2572  LD      L1560
      OUT     Y876
2574  LD      L1561
      OUT     Y877
2576  LD      L1562
      OUT     Y932
2578  LD      L1563
      OUT     Y933
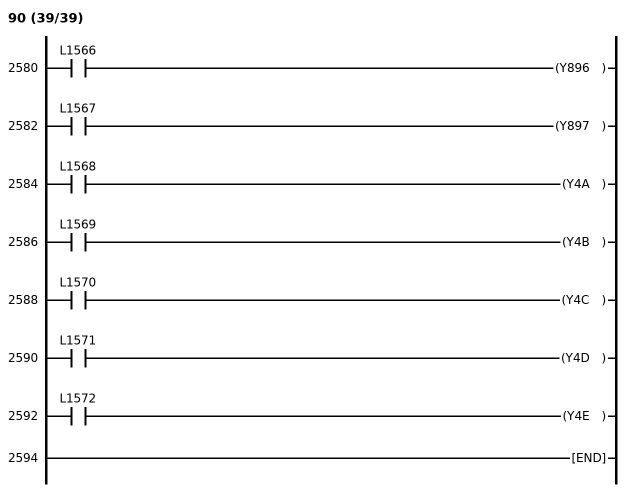
2580  LD      L1566
      OUT     Y896
2582  LD      L1567
      OUT     Y897
2584  LD      L1568
      OUT     Y4A
2586  LD      L1569
      OUT     Y4B
2588  LD      L1570
      OUT     Y4C
2590  LD      L1571
      OUT     Y4D
2592  LD      L1572
      OUT     Y4E
2594  END
END_PROGRAM

PROGRAM 99
0     END
END_PROGRAM

PROGRAM ADVANCE
